FUNCTION "FC_Any_To_Adress" : VOID
TITLE =%version: 0.02 % CN: 30
//Function:
// Reads the start adress of the ANY pointer
//
//History:
//This version  %created_by: nlhdl %
//              %date_created: maandag 7 december 2015 16:01:28 %
//              %release: VI_RAW/RA_Dev %
//
//Modification History:                                   By:    Date:     Rev:
//----------------------------------------------------  -------  --------  -----
//ra#9751: Add source files ECS-P to VI_RAW             nlHdL    14-12-15   0.02
//ra#9751: Add source files ECS-P to VI_RAW             nlHdL    07-12-15   0.02
//7324: ECS-P General from the RD to RA for platform    nlHdL    06-07-15   0.02
//22337: Remove the vibes1.x with the vibes 3.x         nlHdL    09-01-15   0.02
//Initial Revision                                      nlHdL    07-11-13   0.01
//Description:
//Determine the start adress from the ANY pointer
//
FAMILY : VIBES
VERSION : 0.0


VAR_INPUT
  i_ANY_Data : ANY ;	//ANY pointer to Data Record to Retrieve Data from
END_VAR
VAR_OUTPUT
  o_Adress : INT ;	//Adress value of the any pointer
END_VAR
BEGIN
NETWORK
TITLE =AA: Read adress from ANY pointer

      L     P##i_ANY_Data; // 'area-crossing pointer'
      LAR1  ; // Absolute address

      L     W [AR1,P#8.0]; // Adress of the ANY
      SRW   3;
      T     #o_Adress;
END_FUNCTION

